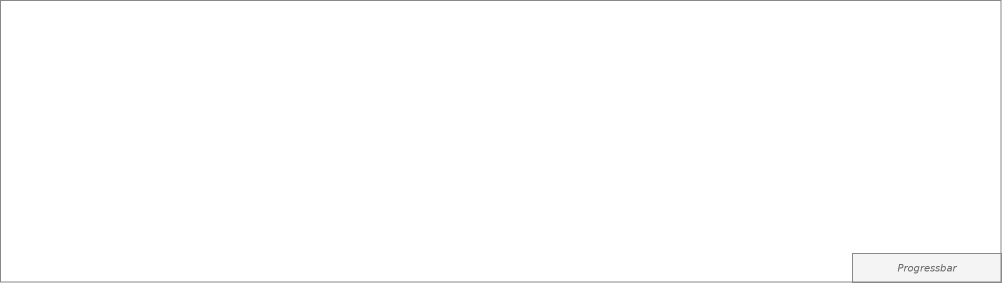
VISUALIZATION Uebersicht  // 1002x283
    Progressbar (852,253 150x30), variable: MAIN.fbStateMachine.timerTON.ET
END_VISUALIZATION

(* stored: Version 1.1.0.1
   Visu Uebersicht: Id {3388f878-4eed-4813-ae35-e96fbec05f25} *)
